// TIA Portal project "Aprenda a Programar CLP do ZERO - André Terra - CLP Fácil" (V15.1)
// Melhorias implementadas no código original das vídeos aulas bonus do curso "Aprenda a Programar CLP do ZERO" do André Terra - CLP Fácil - https://www.clpfacil.com.br

(* hardware
DEVICE "S7-1200 station_1"  S7-1200 Station
   slot 0: "Rack_0"  S7-1200 Rack  Rack  V1.0
   slot 1: "PLC MAIN"  CPU 1215C DC/DC/DC  6ES7 215-1AG40-0XB0  V4.2
*)

// ===== PLC "PLC MAIN"  CPU 1215C DC/DC/DC =====

VAR_GLOBAL   // PLC tag table "Default tag table"
   "Botão Liga B1" AT %I0.0 : Bool;
   "Botão Desliga B2" AT %I0.1 : Bool;
   "Sensor S1" AT %I0.2 : Bool;
   "Sensor S2" AT %I0.3 : Bool;
   "Sensor S3" AT %I0.4 : Bool;
   "Sensor S4" AT %I0.5 : Bool;
   "Motor M1" AT %Q0.0 : Bool;
   "Motor M2" AT %Q0.1 : Bool;
   "Cilindro C1" AT %Q0.2 : Bool;
   "Auxiliar A1" AT %M10.1 : Bool;
   "Auxiliar A2" AT %M10.2 : Bool;
   "Ciclo de Funcionamento" AT %M10.0 : Bool;
END_VAR

// folder: System blocks/Program resources

DATA_BLOCK "IEC_Timer_0_DB"   // DB1
{ S7_Optimized_Access := 'TRUE' }
AUTHOR : Simatic
FAMILY : IEC
NAME : IEC_TMR
VERSION : 1.0
// stored: InstanceOfName IEC_TIMER
"IEC_TIMER"
BEGIN
END_DATA_BLOCK

// folder: (top level)

FUNCTION "Esteira Caixas" : Void   // FC1, LAD
{ S7_Optimized_Access := 'TRUE' }
VERSION : 0.1
BEGIN

REGION Network 1: Liga/Desliga Sistema de Esteiras Caixas (Ciclo de Funcionamento)
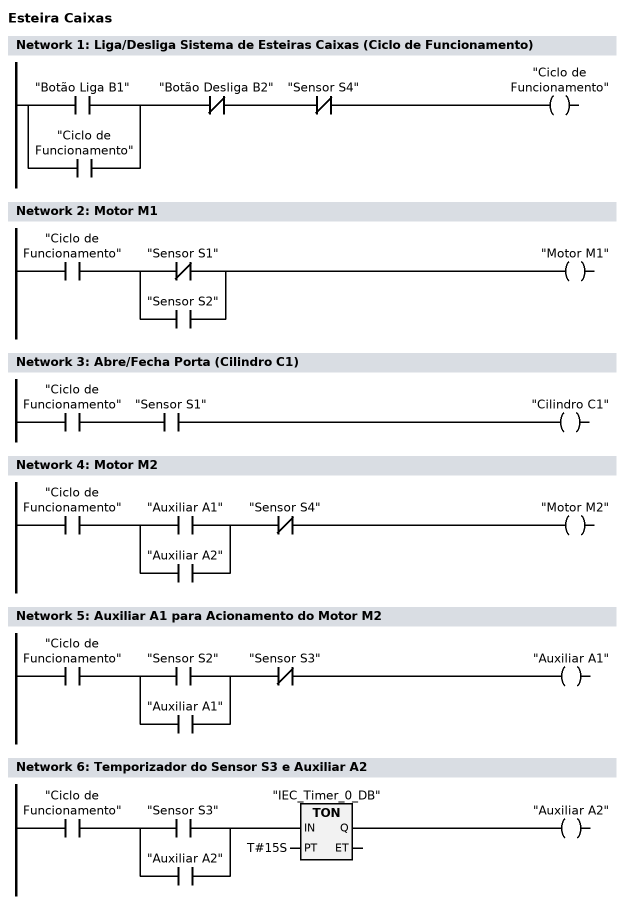
   RUNG wire#powerrail
      Contact( "Botão Liga B1" )
      wire#w1
      I_Contact( "Botão Desliga B2" )
      I_Contact( "Sensor S4" )
      Coil( "Ciclo de Funcionamento" )
   END_RUNG
   RUNG wire#powerrail
      Contact( "Ciclo de Funcionamento" )
   END_RUNG wire#w1
   // the same network as SCL:
   "Ciclo de Funcionamento" := ("Botão Liga B1" OR "Ciclo de Funcionamento") AND NOT "Botão Desliga B2" AND NOT "Sensor S4";
END_REGION

REGION Network 2: Motor M1
   RUNG wire#powerrail
      Contact( "Ciclo de Funcionamento" )
      wire#w1
      I_Contact( "Sensor S1" )
      wire#w2
      Coil( "Motor M1" )
   END_RUNG
   RUNG wire#w1
      Contact( "Sensor S2" )
   END_RUNG wire#w2
   // the same network as SCL:
   "Motor M1" := "Ciclo de Funcionamento" AND (NOT "Sensor S1" OR "Sensor S2");
END_REGION

REGION Network 3: Abre/Fecha Porta (Cilindro C1)
   RUNG wire#powerrail
      Contact( "Ciclo de Funcionamento" )
      Contact( "Sensor S1" )
      Coil( "Cilindro C1" )
   END_RUNG
   // the same network as SCL:
   "Cilindro C1" := "Ciclo de Funcionamento" AND "Sensor S1";
END_REGION

REGION Network 4: Motor M2
   RUNG wire#powerrail
      Contact( "Ciclo de Funcionamento" )
      wire#w1
      Contact( "Auxiliar A1" )
      wire#w2
      I_Contact( "Sensor S4" )
      Coil( "Motor M2" )
   END_RUNG
   RUNG wire#w1
      Contact( "Auxiliar A2" )
   END_RUNG wire#w2
   // the same network as SCL:
   "Motor M2" := "Ciclo de Funcionamento" AND ("Auxiliar A1" OR "Auxiliar A2") AND NOT "Sensor S4";
END_REGION

REGION Network 5: Auxiliar A1 para Acionamento do Motor M2
   RUNG wire#powerrail
      Contact( "Ciclo de Funcionamento" )
      wire#w1
      Contact( "Sensor S2" )
      wire#w2
      I_Contact( "Sensor S3" )
      Coil( "Auxiliar A1" )
   END_RUNG
   RUNG wire#w1
      Contact( "Auxiliar A1" )
   END_RUNG wire#w2
   // the same network as SCL:
   "Auxiliar A1" := "Ciclo de Funcionamento" AND ("Sensor S2" OR "Auxiliar A1") AND NOT "Sensor S3";
END_REGION

REGION Network 6: Temporizador do Sensor S3 e Auxiliar A2
   "IEC_Timer_0_DB".TON(IN := "Ciclo de Funcionamento" AND ("Sensor S3" OR "Auxiliar A2"), PT := T#15S);
   "Auxiliar A2" := "IEC_Timer_0_DB".Q;
END_REGION
END_FUNCTION

ORGANIZATION_BLOCK "Main"   // OB1, LAD, ProgramCycle
TITLE = "Main Program Sweep (Cycle)"
{ S7_Optimized_Access := 'TRUE' }
VERSION : 0.1
   VAR_INPUT
      Initial_Call : Bool;   // Initial call of this OB
      Remanence : Bool;   // =True, if remanent data are available
   END_VAR
BEGIN

REGION Network 1
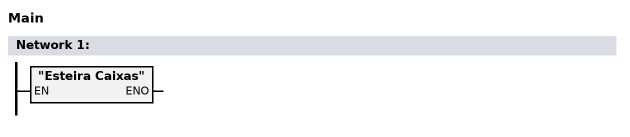
   RUNG wire#powerrail
      "Esteira Caixas"()
   END_RUNG
   // the same network as SCL:
   "Esteira Caixas"();
END_REGION
END_ORGANIZATION_BLOCK